// Mitsubishi GX Works2 project: test   PLC: Q03UDV

PROGRAM MAIN
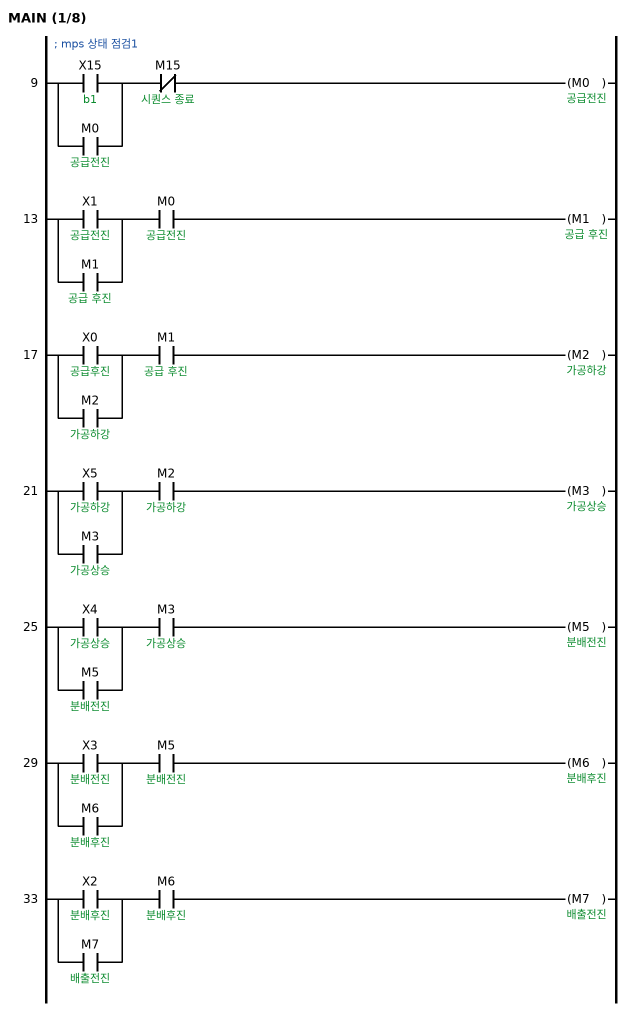
; mps 상태 점검1
9     LD      X15  ; b1
      OR      M0  ; 공급전진
      ANI     M15  ; 시퀀스 종료
      OUT     M0  ; 공급전진
13    LD      X1  ; 공급전진
      OR      M1  ; 공급 후진
      AND     M0  ; 공급전진
      OUT     M1  ; 공급 후진
17    LD      X0  ; 공급후진
      OR      M2  ; 가공하강
      AND     M1  ; 공급 후진
      OUT     M2  ; 가공하강
21    LD      X5  ; 가공하강
      OR      M3  ; 가공상승
      AND     M2  ; 가공하강
      OUT     M3  ; 가공상승
25    LD      X4  ; 가공상승
      OR      M5  ; 분배전진
      AND     M3  ; 가공상승
      OUT     M5  ; 분배전진
29    LD      X3  ; 분배전진
      OR      M6  ; 분배후진
      AND     M5  ; 분배전진
      OUT     M6  ; 분배후진
33    LD      X2  ; 분배후진
      OR      M7  ; 배출전진
      AND     M6  ; 분배후진
      OUT     M7  ; 배출전진
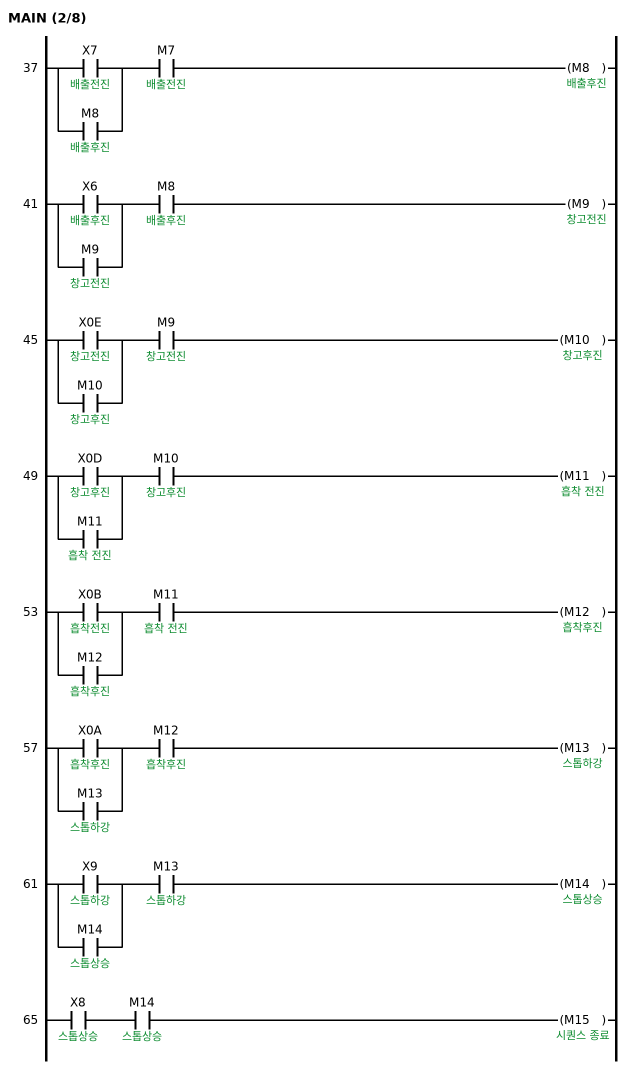
37    LD      X7  ; 배출전진
      OR      M8  ; 배출후진
      AND     M7  ; 배출전진
      OUT     M8  ; 배출후진
41    LD      X6  ; 배출후진
      OR      M9  ; 창고전진
      AND     M8  ; 배출후진
      OUT     M9  ; 창고전진
45    LD      X0E  ; 창고전진
      OR      M10  ; 창고후진
      AND     M9  ; 창고전진
      OUT     M10  ; 창고후진
49    LD      X0D  ; 창고후진
      OR      M11  ; 흡착 전진
      AND     M10  ; 창고후진
      OUT     M11  ; 흡착 전진
53    LD      X0B  ; 흡착전진
      OR      M12  ; 흡착후진
      AND     M11  ; 흡착 전진
      OUT     M12  ; 흡착후진
57    LD      X0A  ; 흡착후진
      OR      M13  ; 스톱하강
      AND     M12  ; 흡착후진
      OUT     M13  ; 스톱하강
61    LD      X9  ; 스톱하강
      OR      M14  ; 스톱상승
      AND     M13  ; 스톱하강
      OUT     M14  ; 스톱상승
65    LD      X8  ; 스톱상승
      AND     M14  ; 스톱상승
      OUT     M15  ; 시퀀스 종료
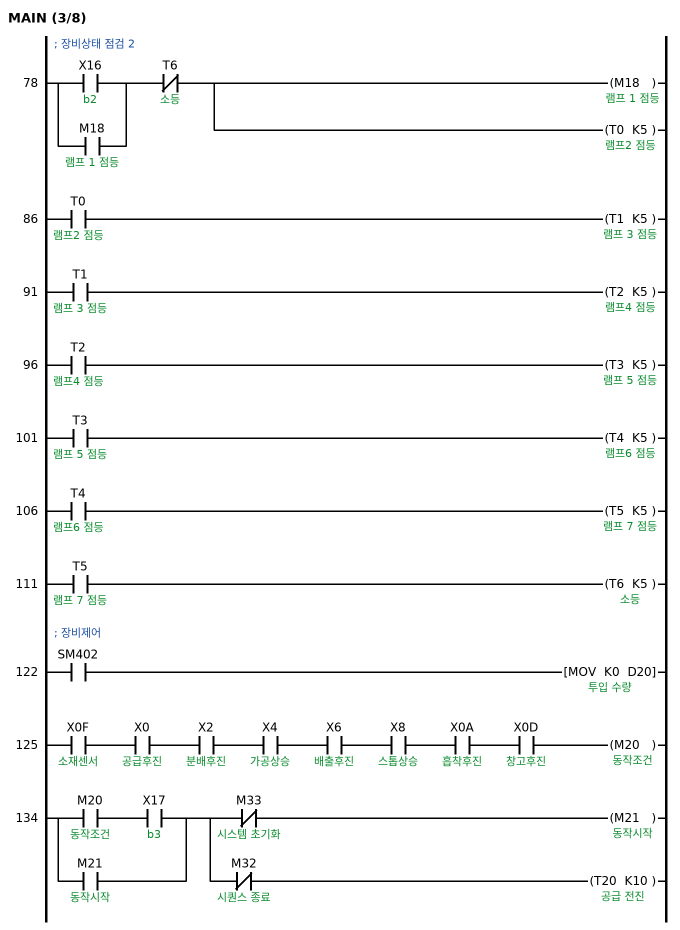
; 장비상태 점검 2
78    LD      X16  ; b2
      OR      M18  ; 램프 1 점등
      ANI     T6  ; 소등
      OUT     M18  ; 램프 1 점등
      OUT     T0 K5  ; 램프2 점등
86    LD      T0  ; 램프2 점등
      OUT     T1 K5  ; 램프 3 점등
91    LD      T1  ; 램프 3 점등
      OUT     T2 K5  ; 램프4 점등
96    LD      T2  ; 램프4 점등
      OUT     T3 K5  ; 램프 5 점등
101   LD      T3  ; 램프 5 점등
      OUT     T4 K5  ; 램프6 점등
106   LD      T4  ; 램프6 점등
      OUT     T5 K5  ; 램프 7 점등
111   LD      T5  ; 램프 7 점등
      OUT     T6 K5  ; 소등
; 장비제어
122   LD      SM402
      MOV     K0 D20  ; 투입 수량
125   LD      X0F  ; 소재센서
      AND     X0  ; 공급후진
      AND     X2  ; 분배후진
      AND     X4  ; 가공상승
      AND     X6  ; 배출후진
      AND     X8  ; 스톱상승
      AND     X0A  ; 흡착후진
      AND     X0D  ; 창고후진
      OUT     M20  ; 동작조건
134   LD      M20  ; 동작조건
      AND     X17  ; b3
      OR      M21  ; 동작시작
      MPS
      ANI     M33  ; 시스템 초기화
      OUT     M21  ; 동작시작
      MPP
      ANI     M32  ; 시퀀스 종료
      OUT     T20 K10  ; 공급 전진
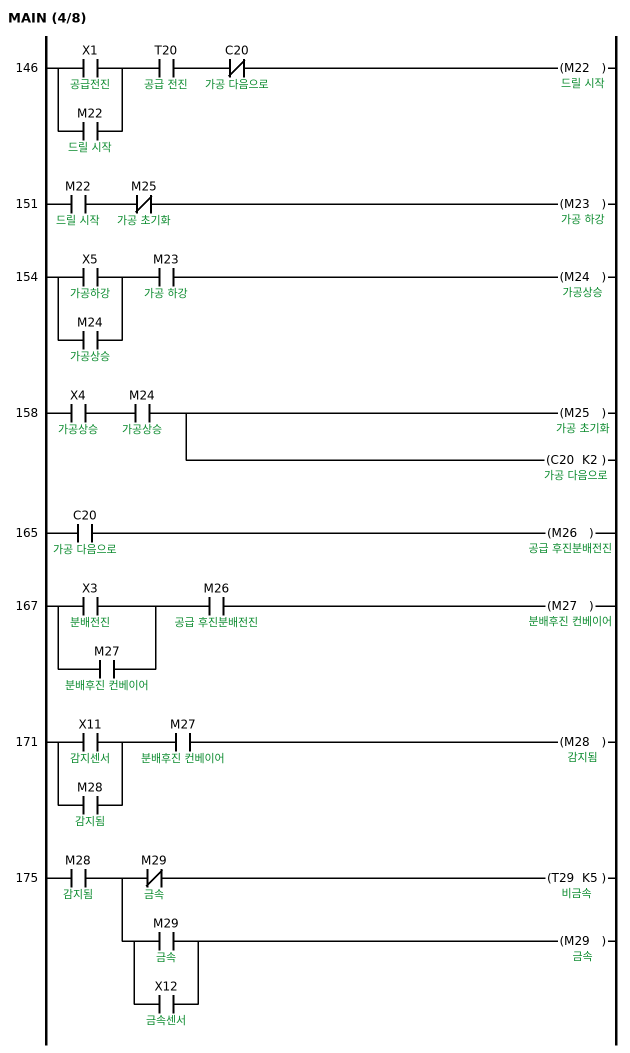
146   LD      X1  ; 공급전진
      OR      M22  ; 드릴 시작
      AND     T20  ; 공급 전진
      ANI     C20  ; 가공 다음으로
      OUT     M22  ; 드릴 시작
151   LD      M22  ; 드릴 시작
      ANI     M25  ; 가공 초기화
      OUT     M23  ; 가공 하강
154   LD      X5  ; 가공하강
      OR      M24  ; 가공상승
      AND     M23  ; 가공 하강
      OUT     M24  ; 가공상승
158   LD      X4  ; 가공상승
      AND     M24  ; 가공상승
      OUT     M25  ; 가공 초기화
      OUT     C20 K2  ; 가공 다음으로
165   LD      C20  ; 가공 다음으로
      OUT     M26  ; 공급 후진분배전진
167   LD      X3  ; 분배전진
      OR      M27  ; 분배후진 컨베이어
      AND     M26  ; 공급 후진분배전진
      OUT     M27  ; 분배후진 컨베이어
171   LD      X11  ; 감지센서
      OR      M28  ; 감지됨
      AND     M27  ; 분배후진 컨베이어
      OUT     M28  ; 감지됨
175   LD      M28  ; 감지됨
      MPS
      ANI     M29  ; 금속
      OUT     T29 K5  ; 비금속
      MPP
      LD      M29  ; 금속
      OR      X12  ; 금속센서
      ANB
      OUT     M29  ; 금속
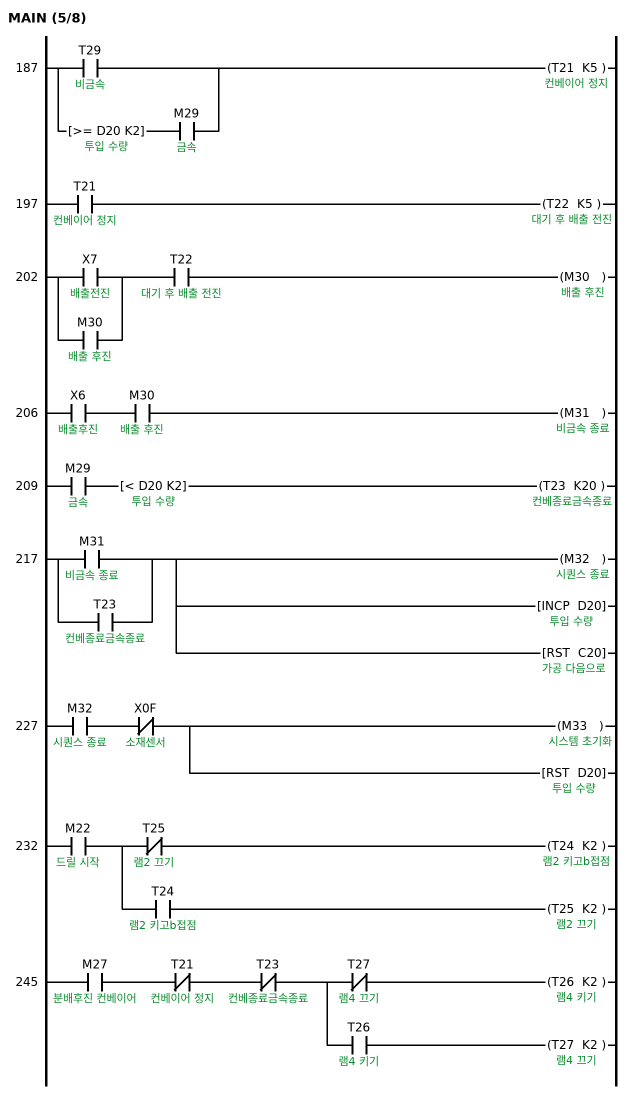
187   LD      T29  ; 비금속
      LD>=    D20 K2  ; 투입 수량
      AND     M29  ; 금속
      ORB
      OUT     T21 K5  ; 컨베이어 정지
197   LD      T21  ; 컨베이어 정지
      OUT     T22 K5  ; 대기 후 배출 전진
202   LD      X7  ; 배출전진
      OR      M30  ; 배출 후진
      AND     T22  ; 대기 후 배출 전진
      OUT     M30  ; 배출 후진
206   LD      X6  ; 배출후진
      AND     M30  ; 배출 후진
      OUT     M31  ; 비금속 종료
209   LD      M29  ; 금속
      AND<    D20 K2  ; 투입 수량
      OUT     T23 K20  ; 컨베종료금속종료
217   LD      M31  ; 비금속 종료
      OR      T23  ; 컨베종료금속종료
      OUT     M32  ; 시퀀스 종료
      INCP    D20
      RST     C20  ; 가공 다음으로
227   LD      M32  ; 시퀀스 종료
      ANI     X0F  ; 소재센서
      OUT     M33  ; 시스템 초기화
      RST     D20  ; 투입 수량
232   LD      M22  ; 드릴 시작
      MPS
      ANI     T25  ; 램2 끄기
      OUT     T24 K2  ; 램2 키고b접점
      MPP
      AND     T24  ; 램2 키고b접점
      OUT     T25 K2  ; 램2 끄기
245   LD      M27  ; 분배후진 컨베이어
      ANI     T21  ; 컨베이어 정지
      ANI     T23  ; 컨베종료금속종료
      MPS
      ANI     T27  ; 램4 끄기
      OUT     T26 K2  ; 램4 키기
      MPP
      AND     T26  ; 램4 키기
      OUT     T27 K2  ; 램4 끄기
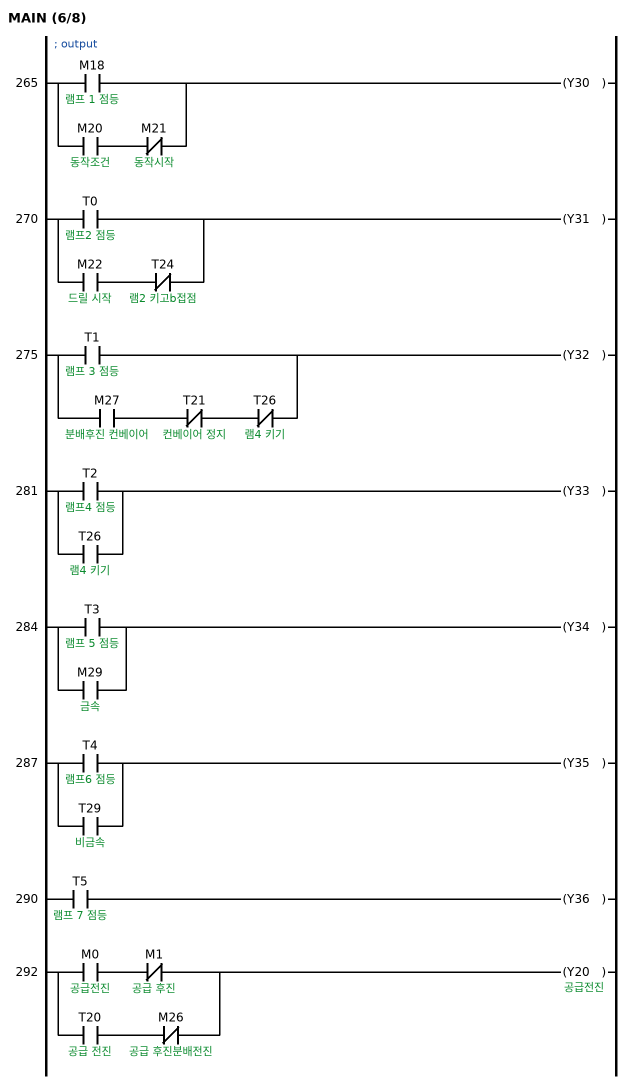
; output
265   LD      M18  ; 램프 1 점등
      LD      M20  ; 동작조건
      ANI     M21  ; 동작시작
      ORB
      OUT     Y30
270   LD      T0  ; 램프2 점등
      LD      M22  ; 드릴 시작
      ANI     T24  ; 램2 키고b접점
      ORB
      OUT     Y31
275   LD      T1  ; 램프 3 점등
      LD      M27  ; 분배후진 컨베이어
      ANI     T21  ; 컨베이어 정지
      ANI     T26  ; 램4 키기
      ORB
      OUT     Y32
281   LD      T2  ; 램프4 점등
      OR      T26  ; 램4 키기
      OUT     Y33
284   LD      T3  ; 램프 5 점등
      OR      M29  ; 금속
      OUT     Y34
287   LD      T4  ; 램프6 점등
      OR      T29  ; 비금속
      OUT     Y35
290   LD      T5  ; 램프 7 점등
      OUT     Y36
292   LD      M0  ; 공급전진
      ANI     M1  ; 공급 후진
      LD      T20  ; 공급 전진
      ANI     M26  ; 공급 후진분배전진
      ORB
      OUT     Y20  ; 공급전진
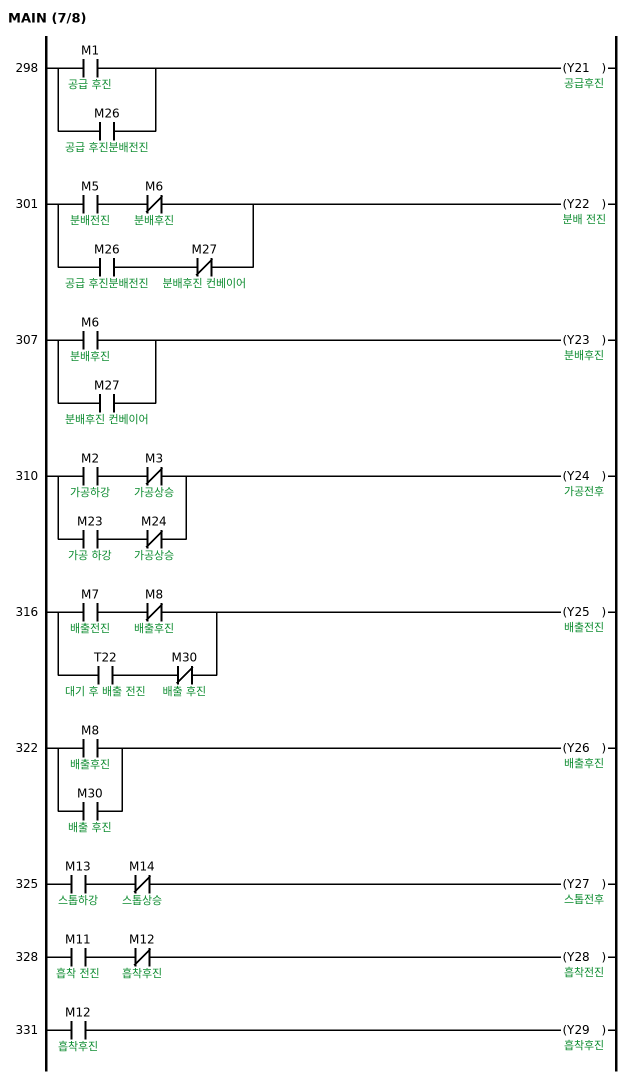
298   LD      M1  ; 공급 후진
      OR      M26  ; 공급 후진분배전진
      OUT     Y21  ; 공급후진
301   LD      M5  ; 분배전진
      ANI     M6  ; 분배후진
      LD      M26  ; 공급 후진분배전진
      ANI     M27  ; 분배후진 컨베이어
      ORB
      OUT     Y22  ; 분배 전진
307   LD      M6  ; 분배후진
      OR      M27  ; 분배후진 컨베이어
      OUT     Y23  ; 분배후진
310   LD      M2  ; 가공하강
      ANI     M3  ; 가공상승
      LD      M23  ; 가공 하강
      ANI     M24  ; 가공상승
      ORB
      OUT     Y24  ; 가공전후
316   LD      M7  ; 배출전진
      ANI     M8  ; 배출후진
      LD      T22  ; 대기 후 배출 전진
      ANI     M30  ; 배출 후진
      ORB
      OUT     Y25  ; 배출전진
322   LD      M8  ; 배출후진
      OR      M30  ; 배출 후진
      OUT     Y26  ; 배출후진
325   LD      M13  ; 스톱하강
      ANI     M14  ; 스톱상승
      OUT     Y27  ; 스톱전후
328   LD      M11  ; 흡착 전진
      ANI     M12  ; 흡착후진
      OUT     Y28  ; 흡착전진
331   LD      M12  ; 흡착후진
      OUT     Y29  ; 흡착후진
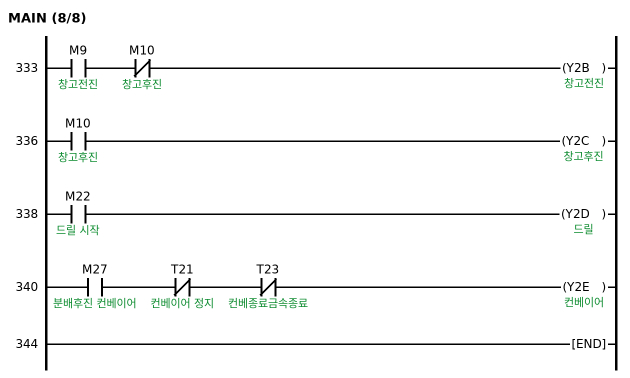
333   LD      M9  ; 창고전진
      ANI     M10  ; 창고후진
      OUT     Y2B  ; 창고전진
336   LD      M10  ; 창고후진
      OUT     Y2C  ; 창고후진
338   LD      M22  ; 드릴 시작
      OUT     Y2D  ; 드릴
340   LD      M27  ; 분배후진 컨베이어
      ANI     T21  ; 컨베이어 정지
      ANI     T23  ; 컨베종료금속종료
      OUT     Y2E  ; 컨베이어
344   END
END_PROGRAM

// device comments not shown above
X0C  ; 흡착여부
X18  ; b4
X19  ; b5
X1A  ; b6
X1B  ; b7
X1C  ; b8
Y2A  ; 흡착작동
